FUNCTION_BLOCK FB_TcExternalTime
VAR
	_hr : HRESULT;
	_ipExtTime : ITcExternalTime;
	_eTimeType: ETcExternalTimeType;
END_VAR

METHOD FB_Exit : BOOL
VAR_INPUT
	bInCopyCode : BOOL; // if TRUE, the exit method is called for exiting an instance that is copied afterwards (online change).
END_VAR
IF _ipExtTime <> 0 THEN
	FW_SafeRelease(ADR(_ipExtTime));
END_IF
END_METHOD

METHOD FB_Init : BOOL
VAR_INPUT
	bInitRetains : BOOL; // if TRUE, the retain variables are initialized (warm start / cold start)
	bInCopyCode : BOOL;  // if TRUE, the instance afterwards gets moved into the copy code (online change)
	eTimeType : ETcExternalTimeType; 
END_VAR
VAR
	ipServer : ITComObjectServer;
END_VAR
ipServer := TwinCAT_SystemInfoVarList._AppInfo.TComSrvPtr;
_eTimeType := eTimeType; 
IF _ipExtTime = 0 THEN
	_hr := ipServer.TcQueryInterface(IID_ITcExternalTime, ADR(_ipExtTime));
	IF FAILED(_hr) THEN RETURN; END_IF
END_IF
END_METHOD

METHOD GetExternalOffset : LINT
VAR_INPUT
END_VAR
IF _ipExtTime <> 0 THEN
	_hr := _ipExtTime.GetExternalTimeOffset(_eTimeType, GetExternalOffset);
	IF _hr <> 0 THEN GetExternalOffset := 0; END_IF
END_IF
END_METHOD

METHOD GetExternalTime : LINT
VAR_INPUT
END_VAR
IF _ipExtTime <> 0 THEN
	GetExternalTime := GetSystemTime();
	_hr := _ipExtTime.SystemTimeToExternalTime(_eTimeType, GetExternalTime);
	IF _hr <> 0 THEN GetExternalTime := 0; END_IF
END_IF
END_METHOD

METHOD GetSystemTime : LINT
GetSystemTime := ULINT_TO_LINT(F_GetSystemTime());
END_METHOD

PROPERTY Result : HRESULT
GET
Result := _hr;
END_GET
END_PROPERTY

END_FUNCTION_BLOCK

(* stored: Version 1.1.0.1, ProductVersion 3.1.4024.0
   POU FB_TcExternalTime: Id {58b70043-1ffe-0feb-250e-d7608868f484}, SpecialFunc None
   Method FB_Exit: Id {304398d5-d409-0352-13f7-e8cf2d8a8a7b}
   Method FB_Init: Id {4c9384c2-8535-05f4-1fb3-c7fedc1b553f}
   Method GetExternalOffset: Id {61f35b05-23d9-0bd3-0194-be60d336bcf3}
   Method GetExternalTime: Id {ea43c81d-c214-0602-2499-9ea7c4beda55}
   Method GetSystemTime: Id {bae1aa72-4dbe-010b-3263-59a242298778}
   Property Result: Id {4d7b6b57-c032-0afa-39dd-669652607c80}
   Get Get: Id {7b126ba8-6963-0854-1e3b-eb392e4dc718} *)
